FUNCTION Convert_BYTE_TO_DWORD : BOOL
VAR_INPUT
	in : BYTE;
	out : REFERENCE TO DWORD;
END_VAR
VAR
	converted : DWORD;
END_VAR

converted := BYTE_TO_DWORD(in);

IF (DWORD_TO_BYTE(converted) <> in) THEN
	RETURN;
END_IF

out := converted;
Convert_BYTE_TO_DWORD := TRUE;

END_FUNCTION

(* stored: Version 1.1.0.1, ProductVersion 3.1.4024.12
   POU Convert_BYTE_TO_DWORD: Id {be9ae90c-1a4d-4dc3-a6f1-db6f2fe3ec29}, SpecialFunc None *)
